// TIA Portal V17 export
// export: Created 2022-12-08T10:21:16.7348916Z, ExportSetting WithDefaults, DisplayName Totally Integrated Automation Portal, DisplayVersion V17 Update 5, DisplayName TIA Portal Openness, DisplayVersion V17 Update 5, DisplayName TIA Portal Version Control Interface, DisplayVersion V17, DisplayName Simotion SCOUT TIA, DisplayVersion 5.4.3.0, DisplayName SINAMICS Startdrive Advanced, DisplayVersion V17 SP1, DisplayName SINAMICS Startdrive G130, G150, S120, S150, SINAMICS MV, S210, DisplayVersion V17 SP1, DisplayName SINAMICS Startdrive G110M, G120, G120C, G120D, G120P, G115D, DisplayVersion V17 SP1, DisplayName STEP 7 Professional, DisplayVersion V17 Update 5, DisplayName STEP 7 Safety, DisplayVersion V17, DisplayName WinCC Advanced, DisplayVersion V17 Update 5
DATA_BLOCK "SERVO"   // DB1300
{ S7_Optimized_Access := 'TRUE' }
VERSION : 0.1
// stored: AutoNumber false, DBAccessibleFromOPCUA true, DBAccessibleFromWebserver true, IsOnlyStoredInLoadMemory false, IsRetainMemResEnabled false, IsWriteProtectedInAS false, MemoryReserve 100
   VAR
      Leimnocken : Array[1..8] of DB_ANY;
      Cam : Array["LOWERAXISNUMBER".."UPPERAXISNUMBER"] of DB_ANY;
      Achse : Array["LOWERAXISNUMBER".."UPPERAXISNUMBER"] of DB_ANY;
   END_VAR
   VAR RETAIN
      AchsMoment : Array["LOWERAXISNUMBER".."UPPERAXISNUMBER"] of "UDT_ServoMoment";
   END_VAR
   VAR
      StatusError : Array["LOWERAXISNUMBER".."UPPERAXISNUMBER"] of "UDT_ServoStatusError";
      ActualData : Array["LOWERAXISNUMBER".."UPPERAXISNUMBER"] of "UDT_ServoActualData";
      StatusError_VM { S7_SetPoint := 'True'} : "UDT_ServoStatusError";
   END_VAR
   VAR RETAIN
      Dynamikwerte { S7_SetPoint := 'True'} : "UDT_ServoData";
      Position_VM { S7_SetPoint := 'True'} : LReal;
   END_VAR
   VAR
      Freigabe : Bool;
   END_VAR
BEGIN
END_DATA_BLOCK
